// Mitsubishi GX Works2 project: v01   PLC: Q02/Q02H

PROGRAM MAIN
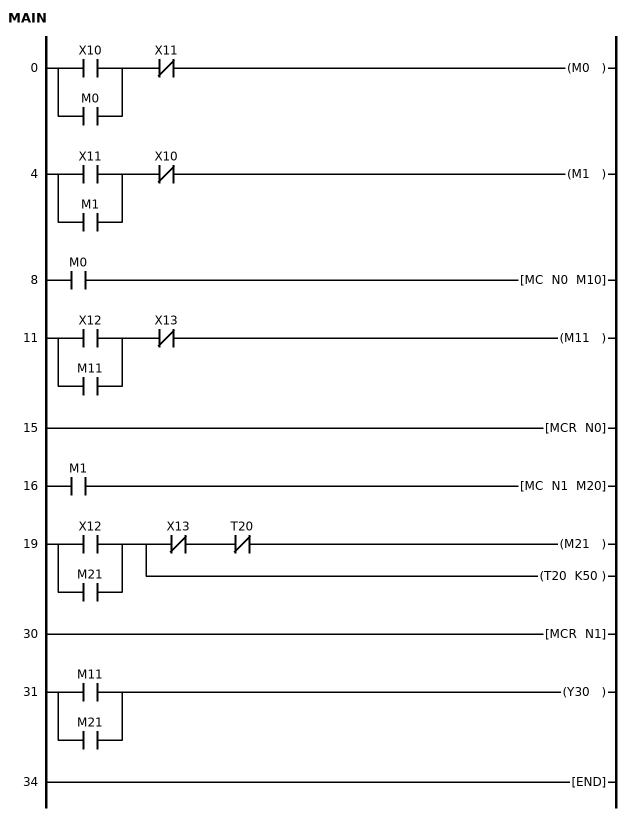
0     LD      X10
      OR      M0
      ANI     X11
      OUT     M0
4     LD      X11
      OR      M1
      ANI     X10
      OUT     M1
8     LD      M0
      MC      N0 M10
11    LD      X12
      OR      M11
      ANI     X13
      OUT     M11
15    MCR     N0
16    LD      M1
      MC      N1 M20
19    LD      X12
      OR      M21
      MPS
      ANI     X13
      ANI     T20
      OUT     M21
      MPP
      OUT     T20 K50
30    MCR     N1
31    LD      M11
      OR      M21
      OUT     Y30
34    END
END_PROGRAM
